FUNCTION_BLOCK DataPanel_xDB_08_DO_SAE_J1939 (* Service Interface Function Block Type *)
  (* Standard: SAE J1939; Function: All Outputs: Digital; Type: DP-40044-05-000; Description: this maps to QX *)
  (* Version 1.0, 2018-12-05, Jose Cabral *)
  (* Version 1.1, 2022-08-04, Franz Hoepfinger, HR Agrartechnik GmbH *)
  (* Version 1.2, 2023-01-05, Franz Hoepfinger, HR Agrartechnik GmbH *)
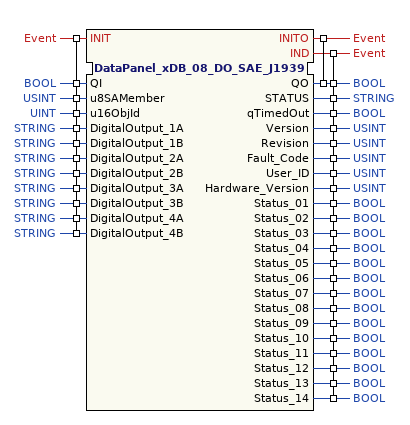
  EVENT_INPUT
    INIT WITH QI, u8SAMember, u16ObjId, DigitalOutput_1A, DigitalOutput_1B, DigitalOutput_2A, DigitalOutput_2B, DigitalOutput_3A, DigitalOutput_3B, DigitalOutput_4A, DigitalOutput_4B; (* Service Initialization *)
  END_EVENT
  EVENT_OUTPUT
    INITO WITH QO; (* Initialization Confirm *)
    IND WITH QO, STATUS, qTimedOut, Version, Revision, Fault_Code, User_ID, Hardware_Version, Status_01, Status_02, Status_03, Status_04, Status_05, Status_06, Status_07, Status_08, Status_09, Status_10, Status_11, Status_12, Status_13, Status_14; (* Indication from Resource *)
  END_EVENT
  VAR_INPUT
    QI : BOOL; (* Event Input Qualifier *)
    u8SAMember : USINT := LO_00; (* Node SA 217..224 *)
    u16ObjId : UINT := ID_NULL; (* Dummy ! set to ID_NULL if in Doubt. ID_OFF deactivates FB. *)
    DigitalOutput_1A : STRING;
    DigitalOutput_1B : STRING;
    DigitalOutput_2A : STRING;
    DigitalOutput_2B : STRING;
    DigitalOutput_3A : STRING;
    DigitalOutput_3B : STRING;
    DigitalOutput_4A : STRING;
    DigitalOutput_4B : STRING;
  END_VAR
  VAR_OUTPUT
    QO : BOOL; (* Event Output Qualifier *)
    STATUS : STRING; (* Service Status *)
    qTimedOut : BOOL;
    Version : USINT;
    Revision : USINT;
    Fault_Code : USINT;
    User_ID : USINT;
    Hardware_Version : USINT;
    Status_01 : BOOL;
    Status_02 : BOOL;
    Status_03 : BOOL;
    Status_04 : BOOL;
    Status_05 : BOOL;
    Status_06 : BOOL;
    Status_07 : BOOL;
    Status_08 : BOOL;
    Status_09 : BOOL;
    Status_10 : BOOL;
    Status_11 : BOOL;
    Status_12 : BOOL;
    Status_13 : BOOL;
    Status_14 : BOOL;
  END_VAR
END_FUNCTION_BLOCK
